(* Logix 5000 project; controller Lab05_anb5567_msw5288 vendor 1 type 14 code 77 rev 20.12; software revision 20.01; part 2 of 2 *)
(* tags used below, declared in another part *)
   simAGT100 : BOOL;   // SIMULATED DEVICE Tank 100 agitator RUN
   simAGT100RNG : BOOL;   // SIMULATED DEVICE Tank 100 agitator RUNNING
   simBV100 : BOOL;   // SIMULATED DEVICE Tank 100 outlet valve
   simBV102 : BOOL;   // SIMULATED DEVICE Tank 100 steam jacket block valve
   simCV101 : BOOL;   // SIMULATED DEVICE Tank 100 water inlet valve
   simCV103 : BOOL;   // SIMULATED DEVICE Tank 100 drain valve
   simCV110 : BOOL;   // SIMULATED DEVICE Tank 100 to line 1 supply valve
   simCV120 : BOOL;   // SIMULATED DEVICE Tank 100 to line 2 supply valve
   simCV130 : BOOL;   // SIMULATED DEVICE Tank 100 to line 3 supply valve
   simCV140 : BOOL;   // SIMULATED DEVICE Tank 100 to line 4 supply valve
   simFCV101 : REAL;   // SIMULATED DEVICE Tank 100 water in steam control valve (% open)
   simFT100 : REAL;   // SIMULATED DEVICE Tank 100 discharge flow rate (gpm)
   simFT101 : REAL;   // SIMULATED DEVICE Tank 100 water in flow rate (gpm)
   simLSH100 : BOOL;   // SIMULATED DEVICE Tank 100 high level switch 1=water at switch
   simLSHH : BOOL;   // SIMULATED DEVICE Tank 100 high-high level switch 1=no water at switch
   simLSL100 : BOOL;   // SIMULATED DEVICE Tank 100 low level switch 1=water at switch
   simLSLL100 : BOOL;   // SIMULATED DEVICE Tank 100 low-low level switch 1=water at switch
   simLT100 : REAL;   // SIMULATED DEVICE Tank 100 level (psi)
   simM101 : BOOL;   // SIMULATED DEVICE Bin 100 screw conveyor RUN
   simM101RNG : BOOL;   // SIMULATED DEVICE Bin 100 screw conveyor RUNNING
   simP100 : BOOL;   // SIMULATED DEVICE Tank 100 outlet pump RUN
   simP100RNG : BOOL;   // SIMULATED DEVICE Tank 100 outlet pump RUNNING
   simPB100A : BOOL;   // SIMULATED DEVICE Start PB 1=pressed
   simPB100B : BOOL;   // SIMULATED DEVICE Stop PB 0=pressed
   simPL100G : BOOL;   // SIMULATED DEVICE Green pilot light
   simPL100R : BOOL;   // SIMULATED DEVICE Red pilot light
   simReal : REAL[100];   // General purpose simulation real numbers
   simSG101 : BOOL;   // SIMULATED DEVICE Bin 100 outlet slide gate
   simSG101CL : BOOL;   // SIMULATED DEVICE Bin 100 outlet slide gate IS CLOSED
   simSG101OP : BOOL;   // SIMULATED DEVICE Bin 100 outlet slide gate IS OPEN
   simSPD100 : REAL;   // SIMULATED DEVICE Tank 100 outlet pump speed command (% fs)
   simSS100 : BOOL;   // SIMULATED DEVICE Enable SS 1=enabled
   simTmr : TIMER[100];   // General purpose simulation timers
   simTT100 : REAL;   // SIMULATED DEVICE Tank 100 product temperature (deg F)
   simTT101 : REAL;   // SIMULATED DEVICE Tank 100 water in temperature (deg F)
   simWT100 : REAL;   // SIMULATED DEVICE Tank 100 weight (lb)
   simWT101 : REAL;   // SIMULATED DEVICE Bin 101 weight (lb)
   FT100 : REAL;   // Tank 100 discharge flow rate (4-20 mA, 0 to 100 gpm)
   FT101 : REAL;   // Tank 100 water in flow rate (4-20 mA, 0 to 150 gpm)
   SimConfig : DINT[100];   // Simulation Configuration Data
   SimLocal_2_I_Data : INT;   // SIMULATED INPUTS 1769-IQ16 Local:2:I
   TT100 : REAL;   // Tank 100 product temperature (4-20 mA, 0 to 250 °F)
   TT101 : REAL;   // Tank 100 water in temperature (4-20 mA, 0 to 250 °F)
(* Simulation, continued *)

ROUTINE MapSimDI   (* ladder *)
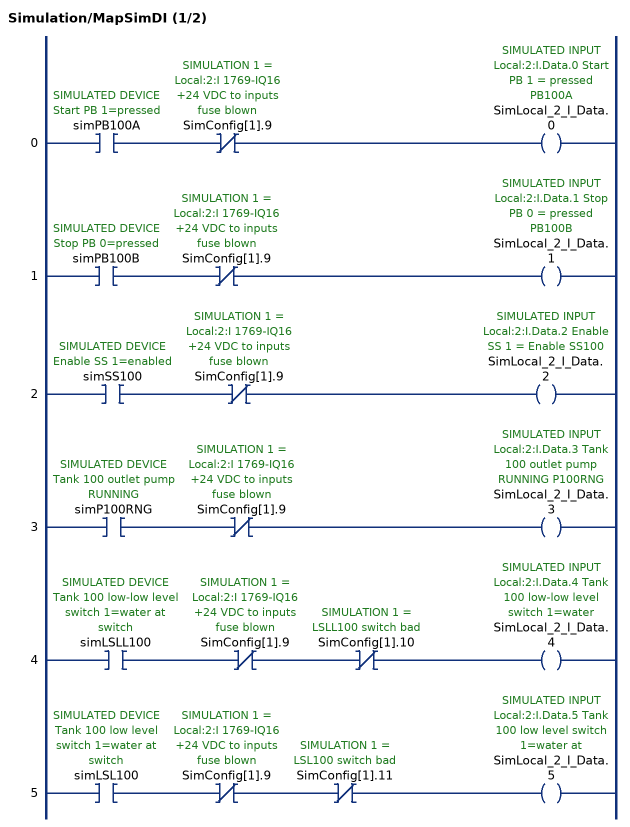
   0: XIC(simPB100A)XIO(SimConfig[1].9)OTE(SimLocal_2_I_Data.0);
   1: XIC(simPB100B)XIO(SimConfig[1].9)OTE(SimLocal_2_I_Data.1);
   2: XIC(simSS100)XIO(SimConfig[1].9)OTE(SimLocal_2_I_Data.2);
   3: XIC(simP100RNG)XIO(SimConfig[1].9)OTE(SimLocal_2_I_Data.3);
   4: XIC(simLSLL100)XIO(SimConfig[1].9)XIO(SimConfig[1].10)OTE(SimLocal_2_I_Data.4);
   5: XIC(simLSL100)XIO(SimConfig[1].9)XIO(SimConfig[1].11)OTE(SimLocal_2_I_Data.5);
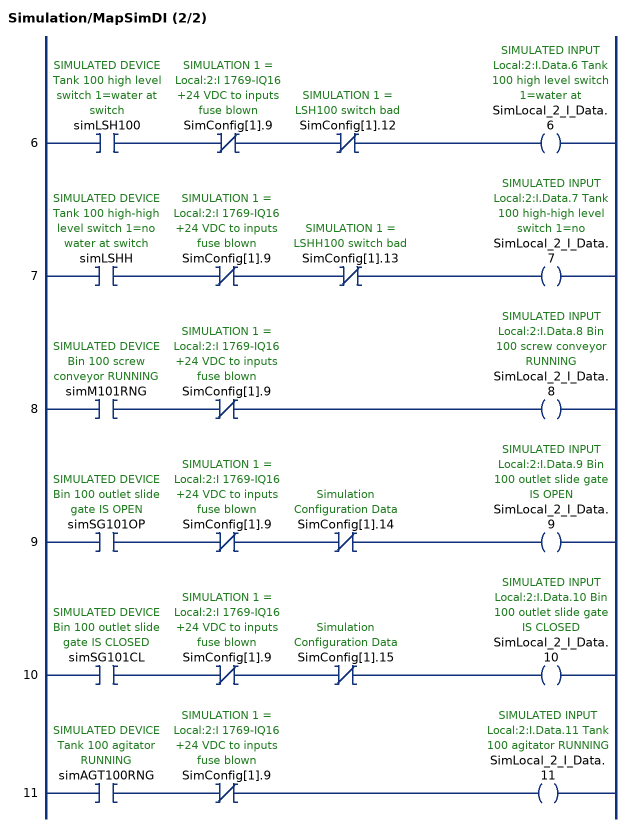
   6: XIC(simLSH100)XIO(SimConfig[1].9)XIO(SimConfig[1].12)OTE(SimLocal_2_I_Data.6);
   7: XIC(simLSHH)XIO(SimConfig[1].9)XIO(SimConfig[1].13)OTE(SimLocal_2_I_Data.7);
   8: XIC(simM101RNG)XIO(SimConfig[1].9)OTE(SimLocal_2_I_Data.8);
   9: XIC(simSG101OP)XIO(SimConfig[1].9)XIO(SimConfig[1].14)OTE(SimLocal_2_I_Data.9);
   10: XIC(simSG101CL)XIO(SimConfig[1].9)XIO(SimConfig[1].15)OTE(SimLocal_2_I_Data.10);
   11: XIC(simAGT100RNG)XIO(SimConfig[1].9)OTE(SimLocal_2_I_Data.11);
END_ROUTINE

ROUTINE MapSimDO   (* ladder *)
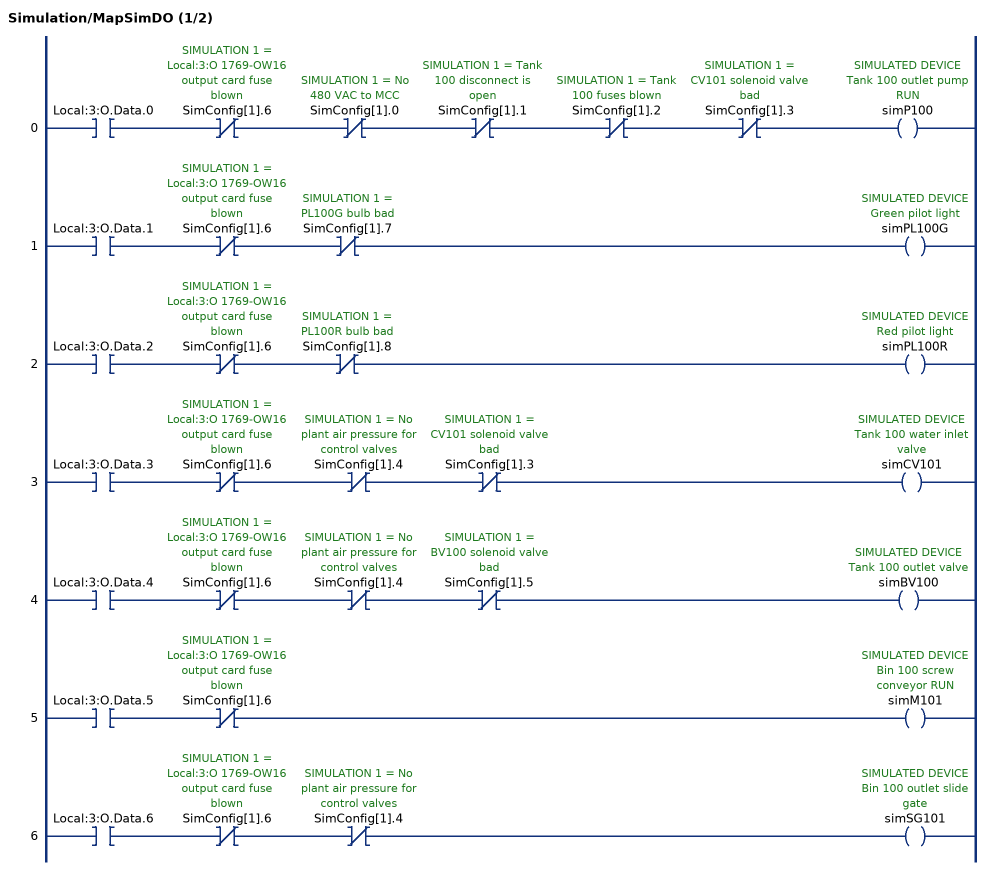
   0: XIC(Local:3:O.Data.0)XIO(SimConfig[1].6)XIO(SimConfig[1].0)XIO(SimConfig[1].1)XIO(SimConfig[1].2)XIO(SimConfig[1].3)OTE(simP100);
   1: XIC(Local:3:O.Data.1)XIO(SimConfig[1].6)XIO(SimConfig[1].7)OTE(simPL100G);
   2: XIC(Local:3:O.Data.2)XIO(SimConfig[1].6)XIO(SimConfig[1].8)OTE(simPL100R);
   3: XIC(Local:3:O.Data.3)XIO(SimConfig[1].6)XIO(SimConfig[1].4)XIO(SimConfig[1].3)OTE(simCV101);
   4: XIC(Local:3:O.Data.4)XIO(SimConfig[1].6)XIO(SimConfig[1].4)XIO(SimConfig[1].5)OTE(simBV100);
   5: XIC(Local:3:O.Data.5)XIO(SimConfig[1].6)OTE(simM101);
   6: XIC(Local:3:O.Data.6)XIO(SimConfig[1].6)XIO(SimConfig[1].4)OTE(simSG101);
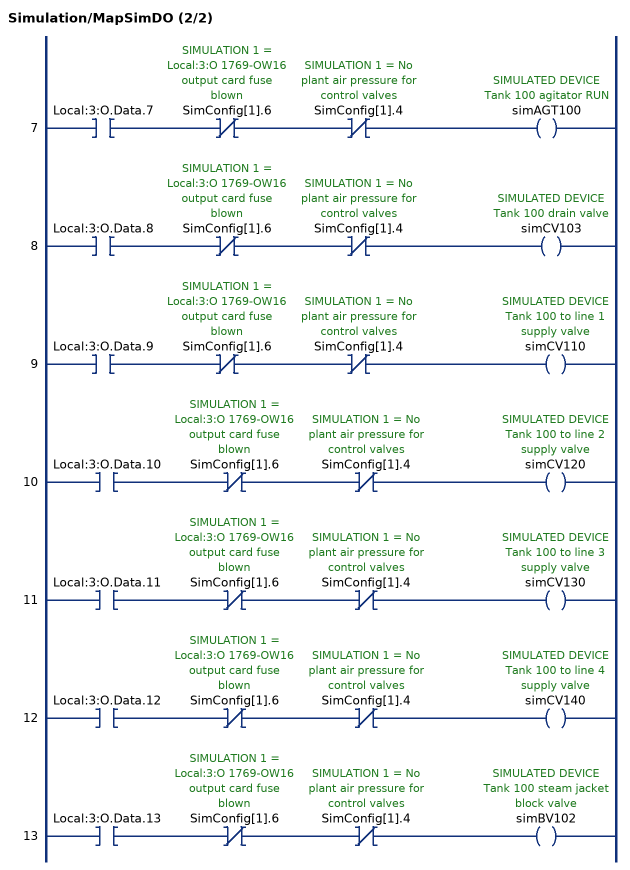
   7: XIC(Local:3:O.Data.7)XIO(SimConfig[1].6)XIO(SimConfig[1].4)OTE(simAGT100);
   8: XIC(Local:3:O.Data.8)XIO(SimConfig[1].6)XIO(SimConfig[1].4)OTE(simCV103);
   9: XIC(Local:3:O.Data.9)XIO(SimConfig[1].6)XIO(SimConfig[1].4)OTE(simCV110);
   10: XIC(Local:3:O.Data.10)XIO(SimConfig[1].6)XIO(SimConfig[1].4)OTE(simCV120);
   11: XIC(Local:3:O.Data.11)XIO(SimConfig[1].6)XIO(SimConfig[1].4)OTE(simCV130);
   12: XIC(Local:3:O.Data.12)XIO(SimConfig[1].6)XIO(SimConfig[1].4)OTE(simCV140);
   13: XIC(Local:3:O.Data.13)XIO(SimConfig[1].6)XIO(SimConfig[1].4)OTE(simBV102);
END_ROUTINE

ROUTINE SimulationLogic   (* ladder *)
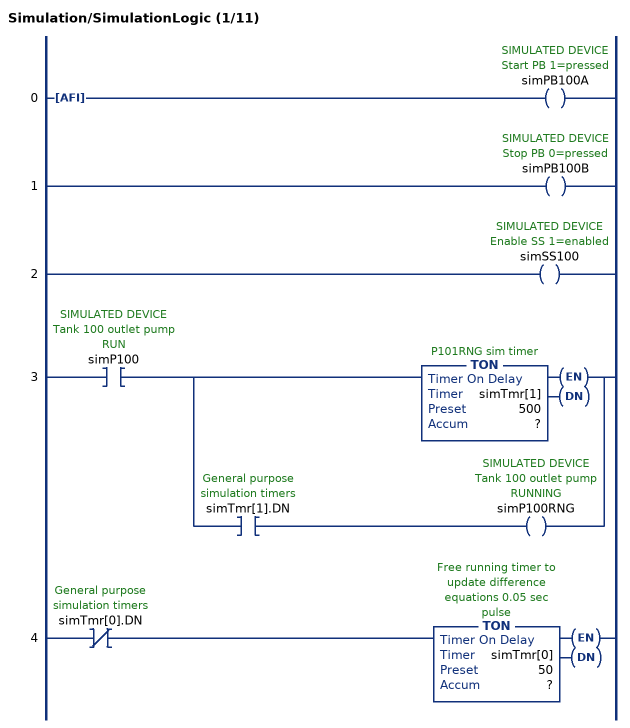
   0: AFI()OTE(simPB100A);
   1: OTE(simPB100B);
   2: OTE(simSS100);
   3: XIC(simP100)[TON(simTmr[1],?,?) ,XIC(simTmr[1].DN) OTE(simP100RNG) ];
   4: XIO(simTmr[0].DN)TON(simTmr[0],?,?);
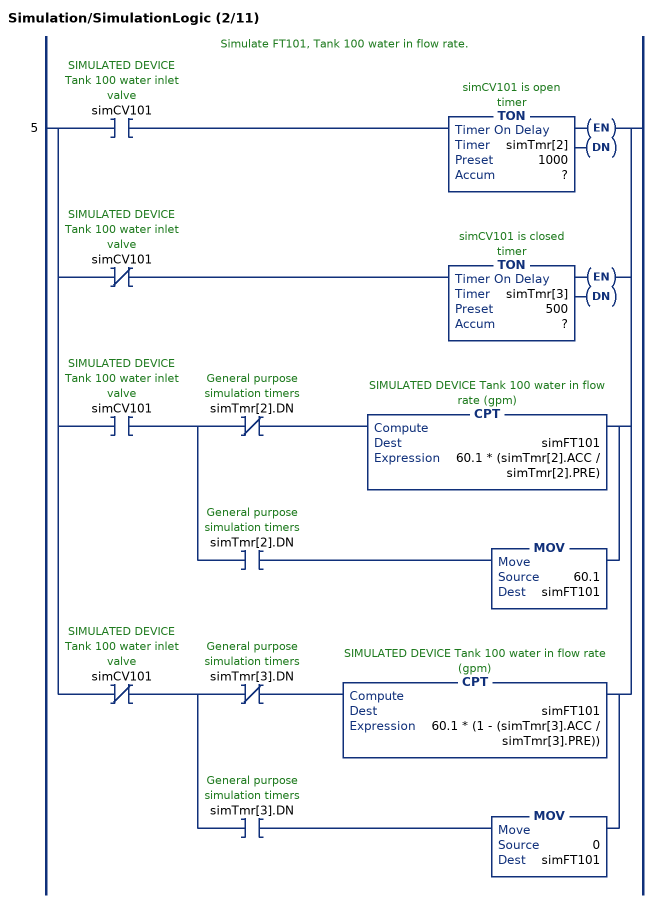
   // Simulate FT101, Tank 100 water in flow rate.
   5: [XIC(simCV101) TON(simTmr[2],?,?) ,XIO(simCV101) TON(simTmr[3],?,?) ,XIC(simCV101) [XIO(simTmr[2].DN) CPT(simFT101,60.1 * (simTmr[2].ACC / simTmr[2].PRE)) ,XIC(simTmr[2].DN) MOV(60.1,simFT101) ] ,XIO(simCV101) [XIO(simTmr[3].DN) CPT(simFT101,60.1 * (1 - (simTmr[3].ACC / simTmr[3].PRE))) ,XIC(simTmr[3].DN) MOV(0,simFT101) ] ];
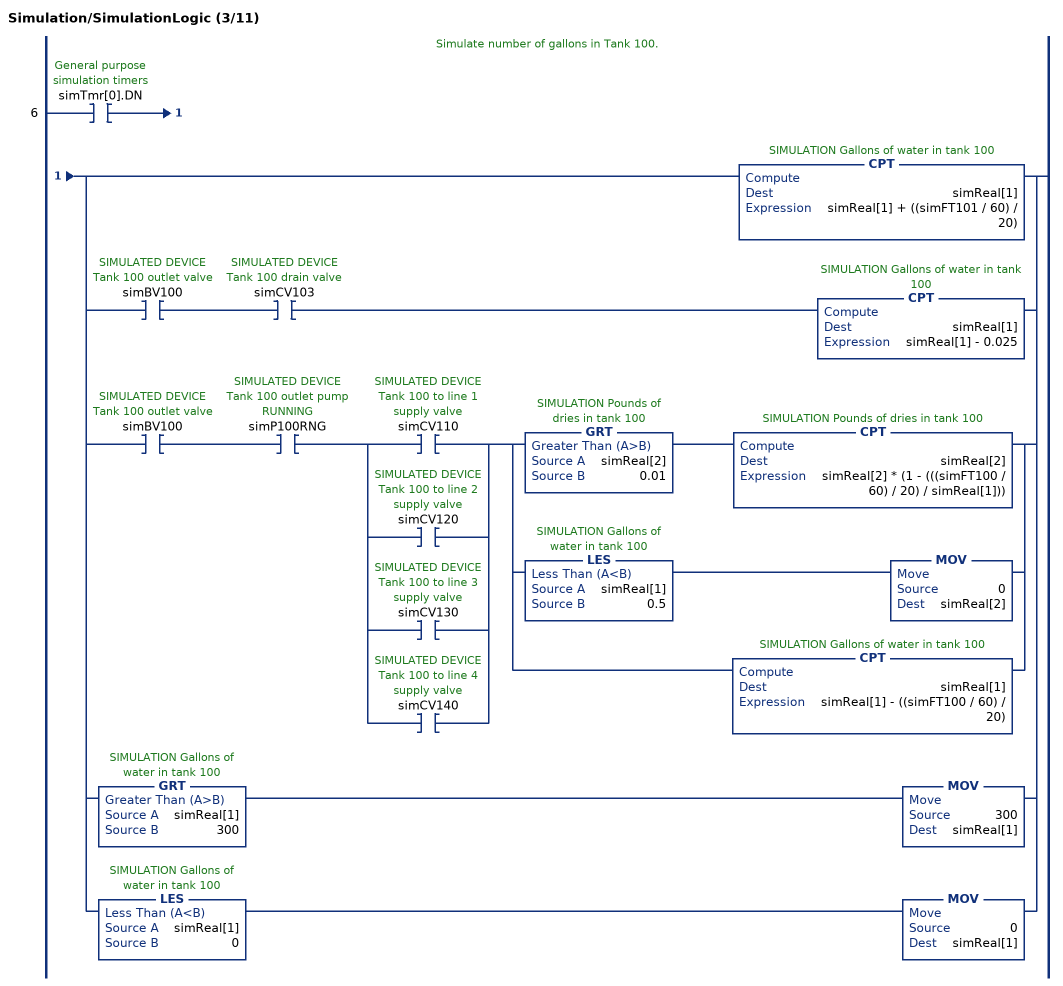
   // Simulate number of gallons in Tank 100.
   6: XIC(simTmr[0].DN)[CPT(simReal[1],simReal[1] + ((simFT101 / 60) / 20)) ,XIC(simBV100) XIC(simCV103) CPT(simReal[1],simReal[1] - 0.025) ,XIC(simBV100) XIC(simP100RNG) [XIC(simCV110) ,XIC(simCV120) ,XIC(simCV130) ,XIC(simCV140) ] [GRT(simReal[2],0.01) CPT(simReal[2],simReal[2] * (1 - (((simFT100 / 60) / 20) / simReal[1]))) ,LES(simReal[1],0.5) MOV(0,simReal[2]) ,CPT(simReal[1],simReal[1] - ((simFT100 / 60) / 20)) ] ,GRT(simReal[1],300) MOV(300,simReal[1]) ,LES(simReal[1],0) MOV(0,simReal[1]) ];
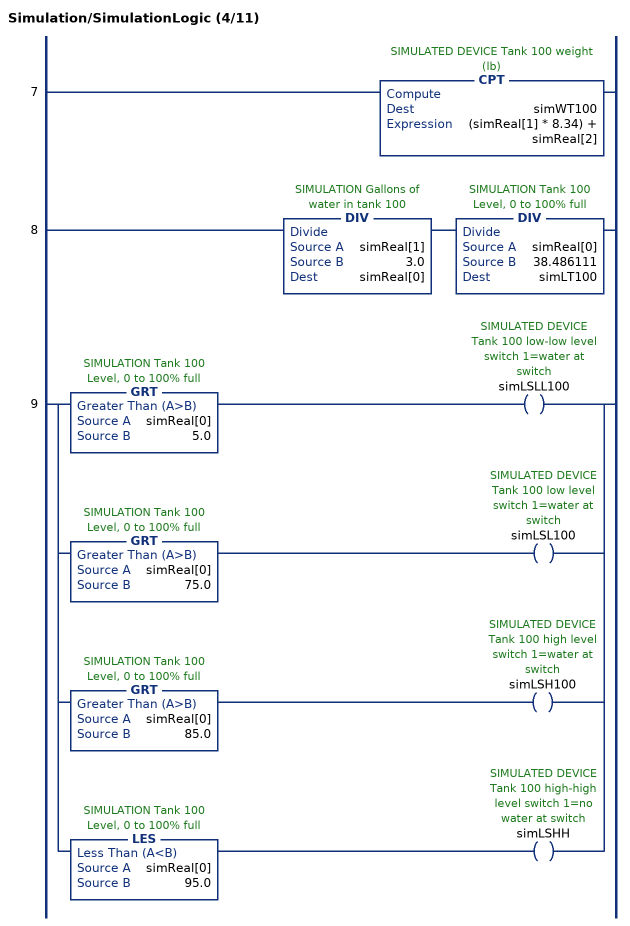
   7: CPT(simWT100,(simReal[1] * 8.34) + simReal[2]);
   8: DIV(simReal[1],3.0,simReal[0])DIV(simReal[0],38.486111,simLT100);
   9: [GRT(simReal[0],5.0) OTE(simLSLL100) ,GRT(simReal[0],75.0) OTE(simLSL100) ,GRT(simReal[0],85.0) OTE(simLSH100) ,LES(simReal[0],95.0) OTE(simLSHH) ];
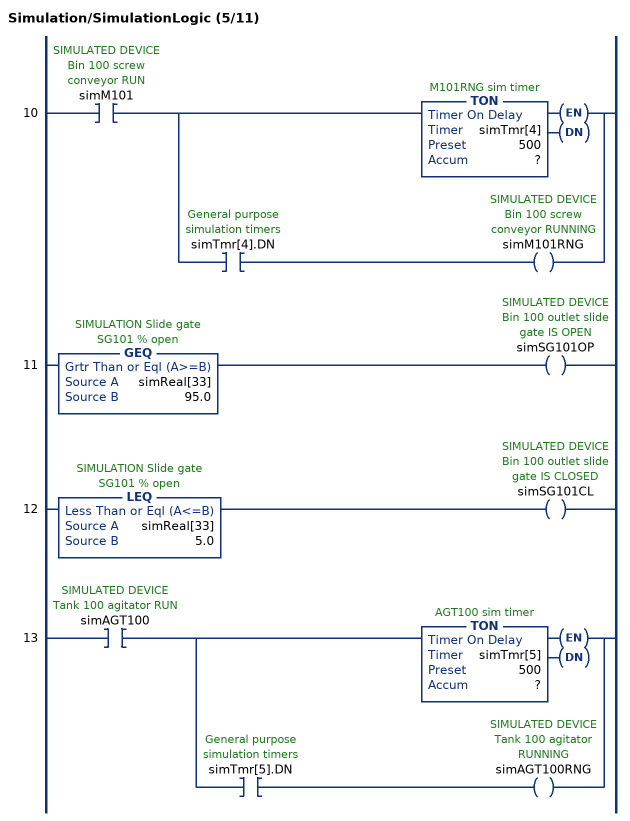
   10: XIC(simM101)[TON(simTmr[4],?,?) ,XIC(simTmr[4].DN) OTE(simM101RNG) ];
   11: GEQ(simReal[33],95.0)OTE(simSG101OP);
   12: LEQ(simReal[33],5.0)OTE(simSG101CL);
   13: XIC(simAGT100)[TON(simTmr[5],?,?) ,XIC(simTmr[5].DN) OTE(simAGT100RNG) ];
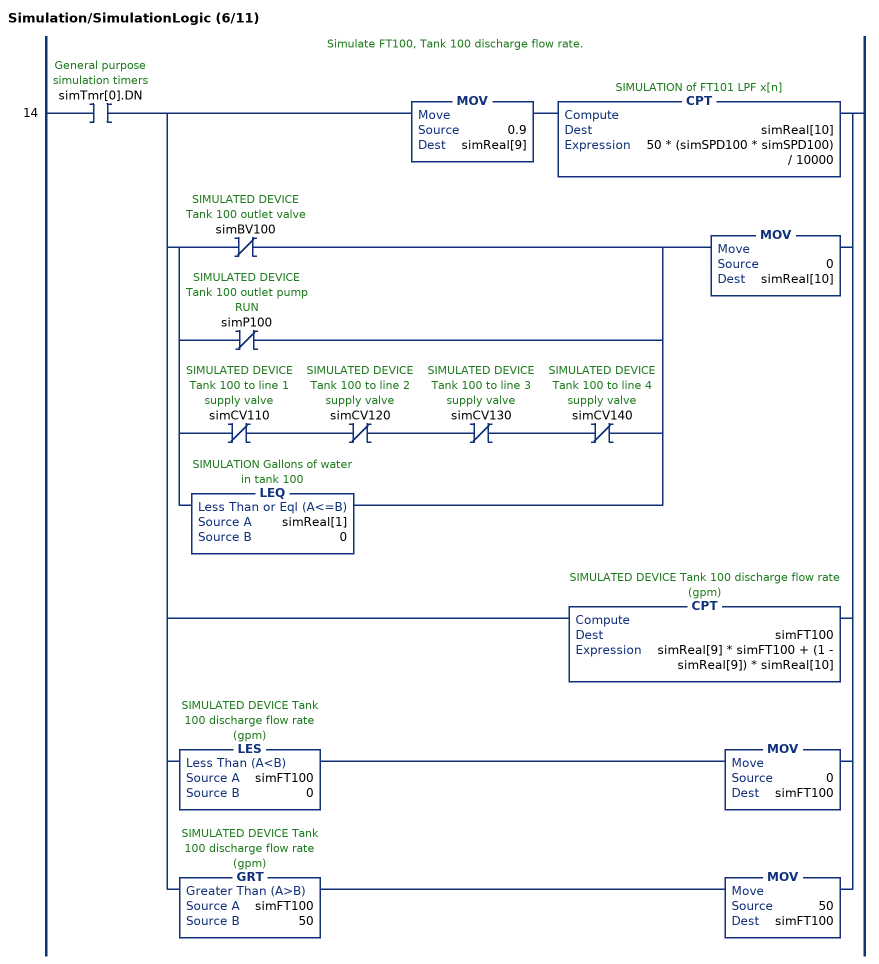
   // Simulate FT100, Tank 100 discharge flow rate.
   14: XIC(simTmr[0].DN)[MOV(0.9,simReal[9]) CPT(simReal[10],50 * (simSPD100 * simSPD100) / 10000) ,[XIO(simBV100) ,XIO(simP100) ,XIO(simCV110) XIO(simCV120) XIO(simCV130) XIO(simCV140) ,LEQ(simReal[1],0) ] MOV(0,simReal[10]) ,CPT(simFT100,simReal[9] * simFT100 + (1 - simReal[9]) * simReal[10]) ,LES(simFT100,0) MOV(0,simFT100) ,GRT(simFT100,50) MOV(50,simFT100) ];
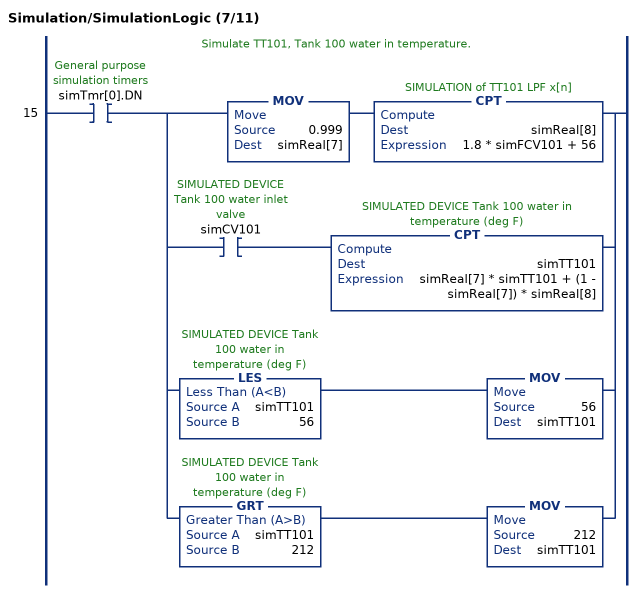
   // Simulate TT101, Tank 100 water in temperature.
   15: XIC(simTmr[0].DN)[MOV(0.999,simReal[7]) CPT(simReal[8],1.8 * simFCV101 + 56) ,XIC(simCV101) CPT(simTT101,simReal[7] * simTT101 + (1 - simReal[7]) * simReal[8]) ,LES(simTT101,56) MOV(56,simTT101) ,GRT(simTT101,212) MOV(212,simTT101) ];
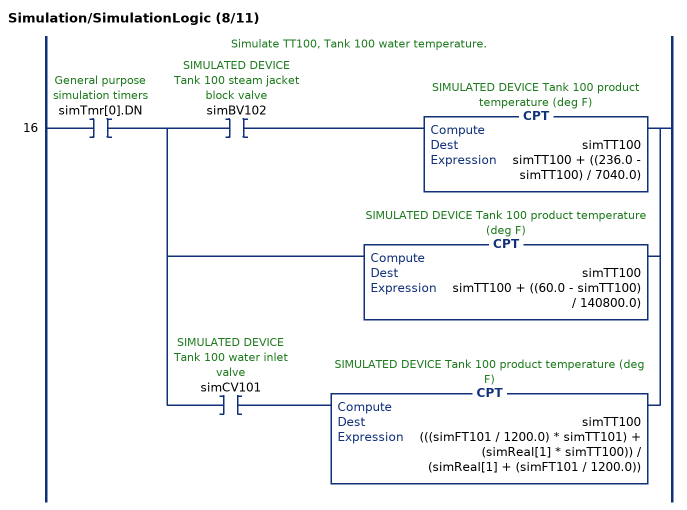
   // Simulate TT100, Tank 100 water temperature.
   16: XIC(simTmr[0].DN)[XIC(simBV102) CPT(simTT100,simTT100 + ((236.0 - simTT100) / 7040.0)) ,CPT(simTT100,simTT100 + ((60.0 - simTT100) / 140800.0)) ,XIC(simCV101) CPT(simTT100,(((simFT101 / 1200.0) * simTT101) + (simReal[1] * simTT100)) / (simReal[1] + (simFT101 / 1200.0))) ];
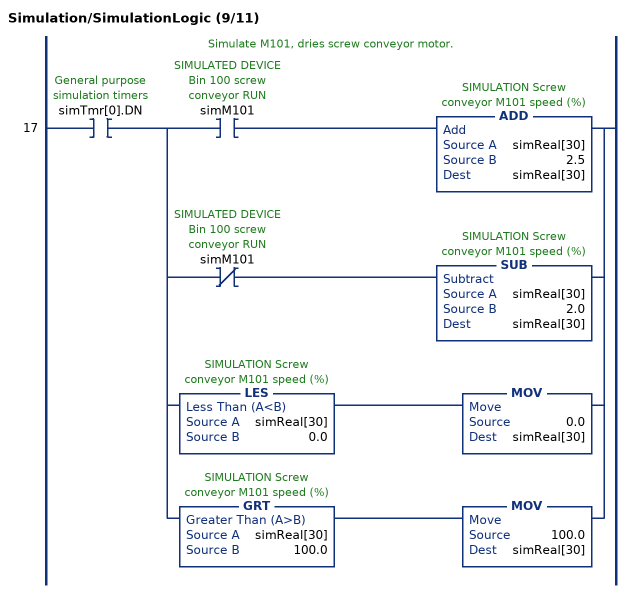
   // Simulate M101, dries screw conveyor motor.
   17: XIC(simTmr[0].DN)[XIC(simM101) ADD(simReal[30],2.5,simReal[30]) ,XIO(simM101) SUB(simReal[30],2.0,simReal[30]) ,LES(simReal[30],0.0) MOV(0.0,simReal[30]) ,GRT(simReal[30],100.0) MOV(100.0,simReal[30]) ];
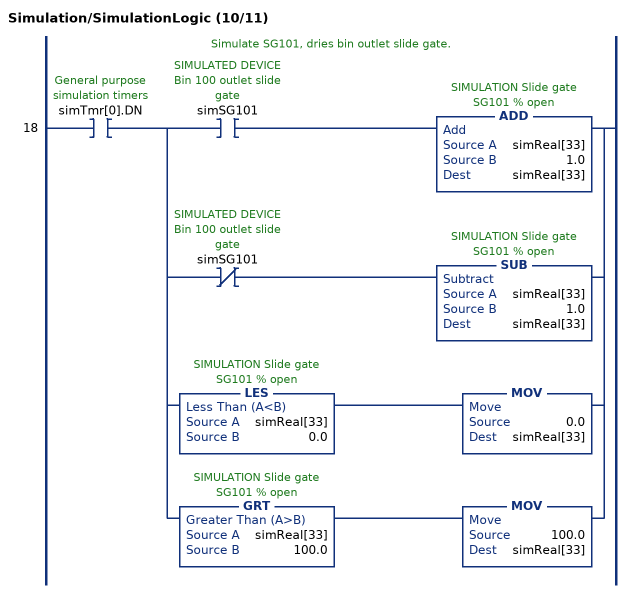
   // Simulate SG101, dries bin outlet slide gate.
   18: XIC(simTmr[0].DN)[XIC(simSG101) ADD(simReal[33],1.0,simReal[33]) ,XIO(simSG101) SUB(simReal[33],1.0,simReal[33]) ,LES(simReal[33],0.0) MOV(0.0,simReal[33]) ,GRT(simReal[33],100.0) MOV(100.0,simReal[33]) ];
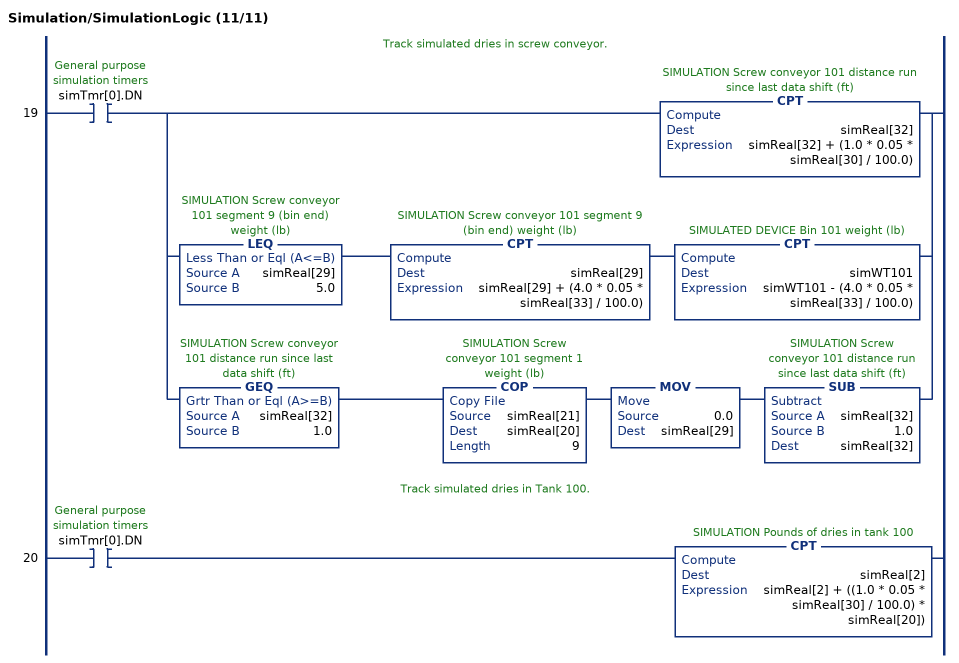
   // Track simulated dries in screw conveyor.
   19: XIC(simTmr[0].DN)[CPT(simReal[32],simReal[32] + (1.0 * 0.05 * simReal[30] / 100.0)) ,LEQ(simReal[29],5.0) CPT(simReal[29],simReal[29] + (4.0 * 0.05 * simReal[33] / 100.0)) CPT(simWT101,simWT101 - (4.0 * 0.05 * simReal[33] / 100.0)) ,GEQ(simReal[32],1.0) COP(simReal[21],simReal[20],9) MOV(0.0,simReal[29]) SUB(simReal[32],1.0,simReal[32]) ];
   // Track simulated dries in Tank 100.
   20: XIC(simTmr[0].DN)CPT(simReal[2],simReal[2] + ((1.0 * 0.05 * simReal[30] / 100.0) * simReal[20]));
END_ROUTINE
END_PROGRAM
